Fanuc KAREL source: kf00044.KL

PROGRAM KF00044
%STACKSIZE=65535
%PRIORITY=65535
%NOLOCKGROUP
VAR
I : INTEGER
J : INTEGER
X : REAL
Y : REAL
B : BOOLEAN
C : BOOLEAN
TXT : STRING[80]
TXT2 : STRING[80]
AI : ARRAY[4] OF INTEGER
BI : ARRAY[4] OF INTEGER
P : XYZWPR
JP : JOINTPOS9
PF : POSITION
STATUS : INTEGER
-- UNRESOLVED DECLARATIONS (source type spelling not recovered)
-- V1 : TYPE_0x0013 (type_u16=0x0013)
-- V2 : TYPE_0x0013 (type_u16=0x0013)
-- REC : TYPE_0x1100 (type_u16=0x1100)
-- REC2 : TYPE_0x1100 (type_u16=0x1100)
BEGIN
REC.VALUE=7
-- UNRESOLVED_PC line 29 opcodes [22 22 30] marker_code=20
END KF00044
